// TIA Portal project "ISA_P8" (V16)

(* hardware
DEVICE "S7-1200 station_1"  S7-1200 Station
   slot 0: "Rack_0"  S7-1200 Rack  Rack  V1.0
   slot 1: "PLC_1"  CPU 1215C DC/DC/DC  6ES7 215-1AG40-0XB0  V4.4
DEVICE "PC-System_1"  SIMATIC PC station
   slot 0: "Estación PC SIMATIC"  Rail  SIMATIC PC-Station  V1.0
      slot 125: "Stationmanager"  Station_Manager  V6.0.4
   slot 1: "HMI_RT_1"  WinCC RT Advanced  6AV2 104-0xxxx-xxxx  16.0.0.0
      slot 33792: "Interfaz del equipo"  Host interface
   slot 2: "IE general_1"  IE General  IE_CP  V8.2.0
*)

// ===== PLC "PLC_1"  CPU 1215C DC/DC/DC =====

VAR_GLOBAL   // PLC tag table "Tabla de variables estándar"
   "Pt100" AT %IW64 : Int;   // Entrada Pt100 en bits
   "System_Byte" AT %MB1 : Byte;
   "FirstScan" AT %M1.0 : Bool;
   "DiagStatusUpdate" AT %M1.1 : Bool;
   "AlwaysTRUE" AT %M1.2 : Bool;
   "AlwaysFALSE" AT %M1.3 : Bool;
   "System_Byte(1)" AT %MB1 : Byte;
   "Pulsador Marcha" AT %I0.0 : Bool;
   "Pulsador Paro" AT %I0.1 : Bool;
   "Resistencia" AT %QW64 : Int;
   "Ventilador" AT %Q0.0 : Bool;
   "Selector_Salida_PID" AT %Q0.1 : Bool;
   "Salida_PWM_PID" AT %Q0.2 : Bool;
END_VAR

DATA_BLOCK "IN_Pt100"   // DB1
{ S7_Optimized_Access := 'TRUE' }
VERSION : 0.1
// stored: InstanceOfName Analog_IN
"Analog_IN"
BEGIN
END_DATA_BLOCK

DATA_BLOCK "Variables"   // DB2
{ S7_Optimized_Access := 'TRUE' }
VERSION : 0.1
   VAR
      Temperatura_Pt100 : Real;   // Temperatura Pt100 en ºC
      Modo_PID : Int;   // Modo de funcionamiento del PID
      Mode_Activate : Bool;   // Activación del modo de funcionamiento del PID
      Flanco_Activate : Bool;   // Flanco de "Mode_Activate"
      Flanco_Paro : Bool;   // Flanco de "Pulsador_Paro"
      Reset_PID : Bool;   // Reset del PID en SCADA
      Salida_PID : Real;   // Salida del PID (0-100)
      Setpoint_PID : Real;   // Setpoint del PID
      Ventilador_SCADA : Bool;   // Activación del ventilador desde SCADA
      Mode_Activate_SCADA : Bool;   // Mode_Activate desde SCADA
      State_PID : Int;   // Modo Activo en el PID
      Error_PID : Bool;   // Indicación de error en PID
      Manual_Value_PID : Real;   // Valor manual PID
      ErrorBits_PID : DWord;   // Código de error PID
      Activar_PWM_SCADA : Bool;
      Salida_PWM_SCADA : Real;
      Salida_PWM_PID : Bool;
      Control_Todo_Nada_On : Bool;
      Salida_Control_TN : Bool;
   END_VAR
BEGIN
END_DATA_BLOCK

DATA_BLOCK "Analog_OUT_DB"   // DB4
{ S7_Optimized_Access := 'TRUE' }
VERSION : 0.1
// stored: InstanceOfName Analog_OUT
"Analog_OUT"
BEGIN
END_DATA_BLOCK

DATA_BLOCK "OUT_Resistencia"   // DB5
{ S7_Optimized_Access := 'TRUE' }
VERSION : 0.1
// stored: InstanceOfName Analog_OUT
"Analog_OUT"
BEGIN
END_DATA_BLOCK

DATA_BLOCK "Telerruptor_DB"   // DB6
{ S7_Optimized_Access := 'TRUE' }
VERSION : 0.1
// stored: InstanceOfName Telerruptor
"Telerruptor"
BEGIN
END_DATA_BLOCK

FUNCTION_BLOCK "Telerruptor"   // FB2, LAD
{ S7_Optimized_Access := 'TRUE' }
VERSION : 0.1
   VAR_INPUT
      Pulsador : Bool;
   END_VAR
   VAR_OUTPUT
      Salida : Bool;
   END_VAR
   VAR
      Flanco : Bool;
      "on/off" : Bool;
      state : Bool;
   END_VAR
   VAR_TEMP   // added for the SCL form of the ladder/FBD networks
      _w1 : Bool;
   END_VAR
BEGIN

REGION Network 1
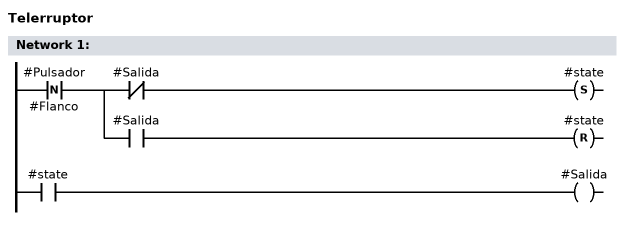
   RUNG wire#powerrail
      N_Contact(operand := #Pulsador, bit := #Flanco)
      wire#w1
      I_Contact( #Salida )
      S_Coil( #state )
   END_RUNG
   RUNG wire#w1
      Contact( #Salida )
      R_Coil( #state )
   END_RUNG
   RUNG wire#powerrail
      Contact( #state )
      Coil( #Salida )
   END_RUNG
   // the same network as SCL:
   #_w1 := NOT #Pulsador AND #Flanco;   // falling edge of #Pulsador
   #Flanco := #Pulsador;
   IF #_w1 AND NOT #Salida THEN #state := TRUE; END_IF;
   IF #_w1 AND #Salida THEN #state := FALSE; END_IF;
   #Salida := #state;
END_REGION
END_FUNCTION_BLOCK

FUNCTION_BLOCK "Analog_IN"   // FB4, LAD
{ S7_Optimized_Access := 'TRUE' }
VERSION : 0.1
   VAR_INPUT
      Input : Int;
      X_min : Real;
      X_max : Real;
      Y_min : Real;
      Y_max : Real;
      IsTension : Bool;
   END_VAR
   VAR_OUTPUT
      Output : Real;
   END_VAR
   VAR
      X_min_bits : Int;
      X_max_bits : Int;
      norm : Real;
   END_VAR
   VAR CONSTANT
      tension_pendent : Real := 2764.8;
      intensity_pendent : Real := 1382.4;
   END_VAR
BEGIN

REGION Network 1 (SCL)

   IF #IsTension THEN
       #X_min_bits := REAL_TO_INT(#X_min * #tension_pendent);
       #X_max_bits := REAL_TO_INT(#X_max * #tension_pendent);
   ELSE
       #X_min_bits := REAL_TO_INT(#X_min * #intensity_pendent);
       #X_max_bits := REAL_TO_INT(#X_max * #intensity_pendent);
   END_IF;
END_REGION

REGION Network 2
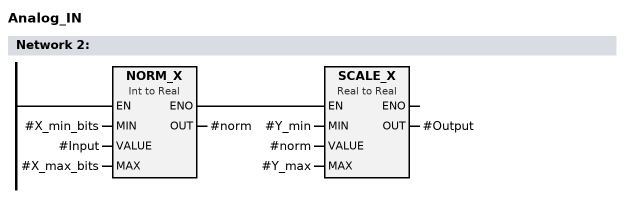
   RUNG wire#powerrail
      { S7_Templates := "[SrcType := Int, DestType := Real]" } Normalize(min := #X_min_bits, value := #Input, max := #X_max_bits, out => #norm)
      { S7_Templates := "[SrcType := Real, DestType := Real]" } Scale(min := #Y_min, value := #norm, max := #Y_max, out => #Output)
   END_RUNG
   // the same network as SCL:
   #norm := NORM_X(MIN := #X_min_bits, VALUE := #Input, MAX := #X_max_bits);
   #Output := SCALE_X(MIN := #Y_min, VALUE := #norm, MAX := #Y_max);
END_REGION
END_FUNCTION_BLOCK

FUNCTION_BLOCK "Analog_OUT"   // FB5, LAD
{ S7_Optimized_Access := 'TRUE' }
VERSION : 0.1
   VAR_INPUT
      Input : Real;
      X_min : Real;
      X_max : Real;
      Y_min : Real;
      Y_max : Real;
      IsTension : Bool;
   END_VAR
   VAR_OUTPUT
      Output : Int;
   END_VAR
   VAR
      Y_min_bits : Int;
      Y_max_bits : Int;
      norm : Real;
   END_VAR
   VAR CONSTANT
      tension_pendent : Real := 2764.8;
      intensity_pendent : Real := 1382.4;
   END_VAR
BEGIN

REGION Network 1 (SCL)

   IF #IsTension THEN
       #Y_min_bits := REAL_TO_INT(#Y_min * #tension_pendent);
       #Y_max_bits := REAL_TO_INT(#Y_max * #tension_pendent);
   ELSE
       #Y_min_bits := REAL_TO_INT(#Y_min * #intensity_pendent);
       #Y_max_bits := REAL_TO_INT(#Y_max * #intensity_pendent);
   END_IF;
END_REGION

REGION Network 2
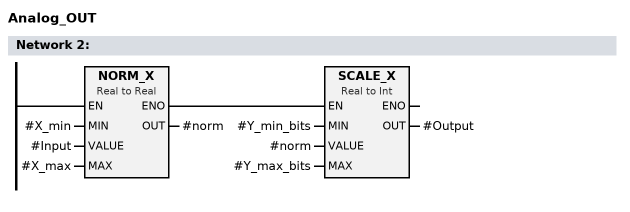
   RUNG wire#powerrail
      { S7_Templates := "[SrcType := Real, DestType := Real]" } Normalize(min := #X_min, value := #Input, max := #X_max, out => #norm)
      { S7_Templates := "[SrcType := Real, DestType := Int]" } Scale(min := #Y_min_bits, value := #norm, max := #Y_max_bits, out => #Output)
   END_RUNG
   // the same network as SCL:
   #norm := NORM_X(MIN := #X_min, VALUE := #Input, MAX := #X_max);
   #Output := SCALE_X(MIN := #Y_min_bits, VALUE := #norm, MAX := #Y_max_bits);
END_REGION
END_FUNCTION_BLOCK

ORGANIZATION_BLOCK "Escalados"   // OB1, LAD, ProgramCycle
TITLE = "Main Program Sweep (Cycle)"
{ S7_Optimized_Access := 'TRUE' }
VERSION : 0.1
   VAR_INPUT
      Initial_Call : Bool;   // Initial call of this OB
      Remanence : Bool;   // =True, if remanent data are available
   END_VAR
BEGIN

REGION Network 1: Escalado acondicionador Pt100
   // Entrada 0-10V del acondicionador de la Pt100 para un rango de 0-100ºC
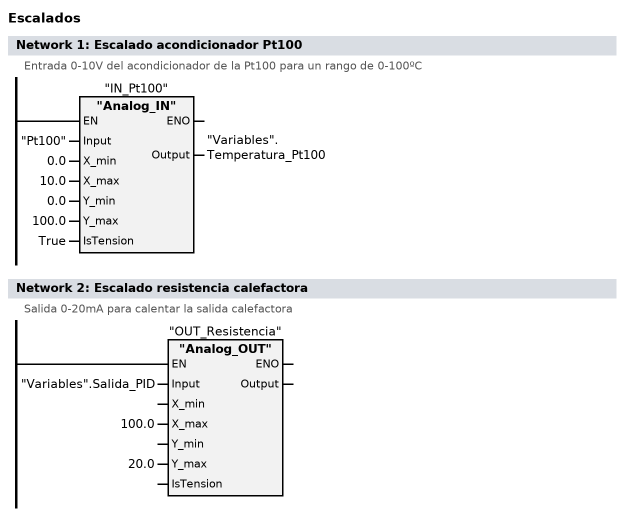
   RUNG wire#powerrail
      "IN_Pt100"(Input := "Pt100", X_min := 0.0, X_max := 10.0, Y_min := 0.0, Y_max := 100.0, IsTension := True, Output => "Variables".Temperatura_Pt100)
   END_RUNG
   // the same network as SCL:
   "IN_Pt100"(Input := "Pt100",   // "Analog_IN"
              X_min := 0.0,
              X_max := 10.0,
              Y_min := 0.0,
              Y_max := 100.0,
              IsTension := True,
              Output => "Variables".Temperatura_Pt100);
END_REGION

REGION Network 2: Escalado resistencia calefactora
   // Salida 0-20mA para calentar la salida calefactora
   RUNG wire#powerrail
      "OUT_Resistencia"(Input := "Variables".Salida_PID, X_min :=, X_max := 100.0, Y_min :=, Y_max := 20.0, IsTension :=, Output =>)
   END_RUNG
   // the same network as SCL:
   "OUT_Resistencia"(Input := "Variables".Salida_PID, X_max := 100.0, Y_max := 20.0);   // "Analog_OUT"
END_REGION

REGION Network 3 (SCL)
   IF "Variables".Salida_PWM_PID THEN
       "Variables".Salida_PWM_SCADA := 100.0;
   ELSE
       "Variables".Salida_PWM_SCADA := 0.0;
   END_IF;
END_REGION
END_ORGANIZATION_BLOCK

ORGANIZATION_BLOCK "PID"   // OB30, LAD, CyclicInterrupt
{ S7_Optimized_Access := 'TRUE' }
VERSION : 0.1
   VAR_INPUT
      Initial_Call : Bool;   // Initial call of this OB
      Event_Count : Int;   // Events discarded
   END_VAR
   VAR_TEMP   // added for the SCL form of the ladder/FBD networks
      _w1 : Bool;
   END_VAR
BEGIN

REGION Network 1: PID
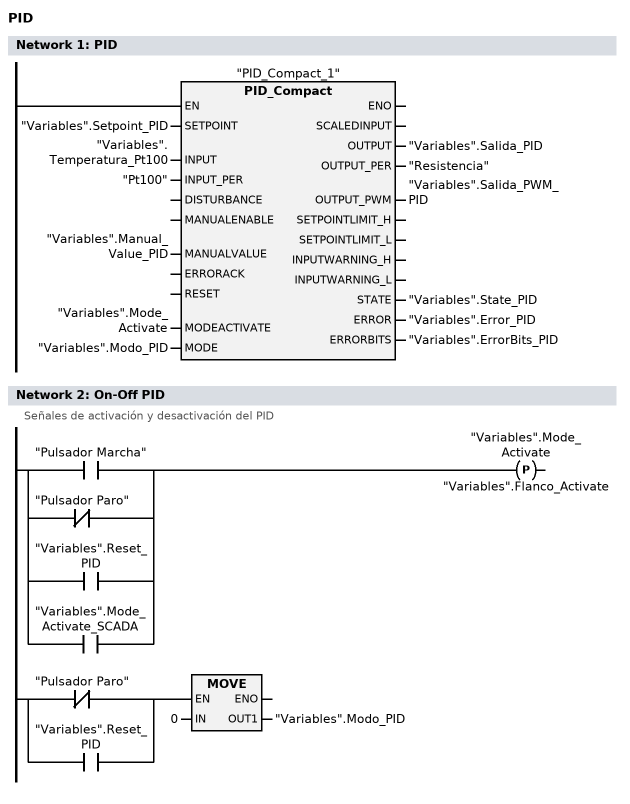
   "PID_Compact_1"(Setpoint := "Variables".Setpoint_PID,   // PID_Compact
                   Input := "Variables".Temperatura_Pt100,
                   Input_PER := "Pt100",
                   ManualValue := "Variables".Manual_Value_PID,
                   ModeActivate := "Variables".Mode_Activate,
                   Mode := "Variables".Modo_PID,
                   Output => "Variables".Salida_PID,
                   Output_PER => "Resistencia",
                   Output_PWM => "Variables".Salida_PWM_PID,
                   State => "Variables".State_PID,
                   Error => "Variables".Error_PID,
                   ErrorBits => "Variables".ErrorBits_PID);
END_REGION

REGION Network 2: On-Off PID
   // Señales de activación y desactivación del PID
   #_w1 := "Pulsador Marcha" OR NOT "Pulsador Paro" OR "Variables".Reset_PID OR "Variables".Mode_Activate_SCADA;
   "Variables".Mode_Activate := #_w1 AND NOT "Variables".Flanco_Activate;   // rising edge
   "Variables".Flanco_Activate := #_w1;
   IF NOT "Pulsador Paro" OR "Variables".Reset_PID THEN "Variables".Modo_PID := 0; END_IF;
END_REGION

REGION Network 3 (SCL)
   "PID_Compact_1".Config.InputPerOn := TRUE;
END_REGION
END_ORGANIZATION_BLOCK

ORGANIZATION_BLOCK "Salidas"   // OB123, LAD, ProgramCycle
TITLE = "Main Program Sweep (Cycle)"
{ S7_Optimized_Access := 'TRUE' }
VERSION : 0.1
   VAR_INPUT
      Initial_Call : Bool;   // Initial call of this OB
      Remanence : Bool;   // =True, if remanent data are available
   END_VAR
BEGIN

REGION Network 1: On-Off Ventilador
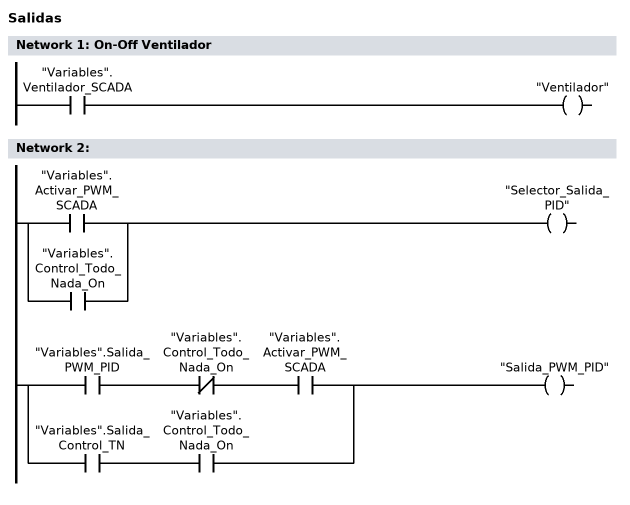
   RUNG wire#powerrail
      Contact( "Variables".Ventilador_SCADA )
      Coil( "Ventilador" )
   END_RUNG
   // the same network as SCL:
   "Ventilador" := "Variables".Ventilador_SCADA;
END_REGION

REGION Network 2
   RUNG wire#powerrail
      Contact( "Variables".Activar_PWM_SCADA )
      wire#w1
      Coil( "Selector_Salida_PID" )
   END_RUNG
   RUNG wire#powerrail
      Contact( "Variables".Control_Todo_Nada_On )
   END_RUNG wire#w1
   RUNG wire#powerrail
      Contact( "Variables".Salida_PWM_PID )
      I_Contact( "Variables".Control_Todo_Nada_On )
      Contact( "Variables".Activar_PWM_SCADA )
      wire#w2
      Coil( "Salida_PWM_PID" )
   END_RUNG
   RUNG wire#powerrail
      Contact( "Variables".Salida_Control_TN )
      Contact( "Variables".Control_Todo_Nada_On )
   END_RUNG wire#w2
   // the same network as SCL:
   "Selector_Salida_PID" := "Variables".Activar_PWM_SCADA OR "Variables".Control_Todo_Nada_On;
   "Salida_PWM_PID" := ("Variables".Salida_PWM_PID AND NOT "Variables".Control_Todo_Nada_On AND "Variables".Activar_PWM_SCADA) OR ("Variables".Salida_Control_TN AND "Variables".Control_Todo_Nada_On);
END_REGION
END_ORGANIZATION_BLOCK

ORGANIZATION_BLOCK "Control_Todo_Nada"   // OB124, SCL, ProgramCycle
TITLE = "Main Program Sweep (Cycle)"
{ S7_Optimized_Access := 'TRUE' }
VERSION : 0.1
   VAR_INPUT
      Initial_Call : Bool;   // Initial call of this OB
      Remanence : Bool;   // =True, if remanent data are available
   END_VAR
BEGIN
   IF "Variables".Temperatura_Pt100 >= "Variables".Setpoint_PID THEN
       "Variables".Salida_Control_TN := FALSE;
   ELSE
       "Variables".Salida_Control_TN := TRUE;
   END_IF;
END_ORGANIZATION_BLOCK

(* ===== HMI "HMI_RT_1" =====
system functions are stored by id; their names below are inferred from use
connection "HMI_Conexión_1": ETHERNET, S7_1200_OMS

HMI tags "Tabla de variables estándar"
   "Variables_Temperatura_Pt100" : Real = PLC Variables.Temperatura_Pt100, 1 s
   "Variables_Modo_PID" : Int = PLC Variables.Modo_PID, 1 s
   "Variables_Ventilador_SCADA" : Bool = PLC Variables.Ventilador_SCADA, 1 s
   "Variables_Setpoint_PID" : Real = PLC Variables.Setpoint_PID, 1 s
   "Variables_Mode_Activate_SCADA" : Bool = PLC Variables.Mode_Activate_SCADA, 1 s
   "Variables_Reset_PID" : Bool = PLC Variables.Reset_PID, 1 s
   "Variables_Salida_PID" : Real = PLC Variables.Salida_PID, 1 s
   "Variables_Error_PID" : Bool = PLC Variables.Error_PID, 1 s
   "Variables_Manual_Value_PID" : Real = PLC Variables.Manual_Value_PID, 1 s
   "Variables_State_PID" : Int = PLC Variables.State_PID, 1 s
   "Variables_ErrorBits_PID" : DWord = PLC Variables.ErrorBits_PID, 1 s
   "PID_Compact_1_Retain_CtrlParams_Gain" : Real = PLC PID_Compact_1.Retain.CtrlParams.Gain, 1 s
   "PID_Compact_1_Retain_CtrlParams_Ti" : Real = PLC PID_Compact_1.Retain.CtrlParams.Ti, 1 s
   "PID_Compact_1_Retain_CtrlParams_Td" : Real = PLC PID_Compact_1.Retain.CtrlParams.Td, 1 s
   "Variables_Activar_PWM_SCADA" : Bool = PLC Variables.Activar_PWM_SCADA, 1 s
   "Variables_Salida_PWM_SCADA" : Real = PLC Variables.Salida_PWM_SCADA, 1 s
   "PID_Compact_1_Retain_CtrlParams_Cycle" : Real = PLC PID_Compact_1.Retain.CtrlParams.Cycle, 1 s
   "PID_Compact_1_Config_MinimumOnTime" : Real = PLC PID_Compact_1.Config.MinimumOnTime, 1 s
   "PID_Compact_1_Config_MinimumOffTime" : Real = PLC PID_Compact_1.Config.MinimumOffTime, 1 s
   "Variables_Control_Todo_Nada_On" : Bool = PLC Variables.Control_Todo_Nada_On, 1 s

text list "Modos_PID": 1 'Optimización Inicial'; 2 'Optimización Fina Manual'; 3 'Modo Automático'; 4 'Modo Manual'

screen "Imagen_1" 800x600
   IOField "Campo ES_1" at 140,209 size 96x32; FormatPattern 999.99; Unit ºC
      ProcessValue <- "Variables_Temperatura_Pt100"
   SymbolicIOField "Campo ES simbólico_1" at 26,530 size 216x32; TextOff '0'; TextOn '1'; TextList "Modos_PID"
      ProcessValue <- "Variables_Modo_PID"
   GraphicView "Visor de gráficos_1" at 254,33 size 251x520; Picture "Captura de pantalla 2023-12-13 131257"
   IOField "Campo ES_2" at 140,123 size 96x32; FormatPattern 99.99
      ProcessValue <- "Variables_Setpoint_PID"
   Button "Botón_1" at 111,42 size 121x32; TextOff 'Ventilador'
      on Click: InvertBit("Variables_Ventilador_SCADA")
   Button "Botón_3" at 146,471 size 96x32; TextOff 'Activate'
      on Press: SetBit("Variables_Mode_Activate_SCADA")
      on Release: ResetBit("Variables_Mode_Activate_SCADA")
   Button "Botón_2" at 26,471 size 96x32; TextOff 'Stop'
      on Press: SetBit("Variables_Reset_PID")
      on Release: ResetBit("Variables_Reset_PID")
   IOField "Campo ES_3" at 519,177 size 96x32; FormatPattern 999.99
      ProcessValue <- "Variables_Salida_PID"
   IOField "Campo ES_4" at 519,400 size 96x32; FormatPattern 9
      ProcessValue <- "Variables_State_PID"
   Rectangle "Rectángulo_1" at 518,436 size 96x20
      Appearance <- "Variables_Error_PID"
   IOField "Campo ES_5" at 140,325 size 96x32; FormatPattern 999.99
      ProcessValue <- "Variables_Manual_Value_PID"
   IOField "Campo ES_6" at 653,25 size 96x32; FormatPattern 99.99
      ProcessValue <- "PID_Compact_1_Retain_CtrlParams_Gain"
   TextField "Campo de texto_1" at 620,29 size 22x22; Text 'k'
   Button "Botón_4" at 652,541 size 96x32; TextOff 'Gráficos'
      on Click: ActivateScreen("Imagen_2", 0)
   IOField "Campo ES_7" at 653,74 size 96x32; FormatPattern 999.99
      ProcessValue <- "PID_Compact_1_Retain_CtrlParams_Ti"
   TextField "Campo de texto_2" at 620,78 size 30x22; Text 'Ti'
   IOField "Campo ES_8" at 653,123 size 96x32; FormatPattern 99.99
      ProcessValue <- "PID_Compact_1_Retain_CtrlParams_Td"
   TextField "Campo de texto_3" at 620,127 size 31x22; Text 'Td'
   IOField "Campo ES_9" at 518,462 size 98x32; FormatPattern FFFF
      ProcessValue <- "Variables_ErrorBits_PID"
   Switch "Interruptor_1" at 642,214 size 120x88; CaptionText 'Salida PWM'; TextOff 'OFF'; TextOn 'ON'
      ProcessValue <- "Variables_Activar_PWM_SCADA"
   IOField "Campo ES_10" at 651,353 size 96x32; FormatPattern 99.99
      ProcessValue <- "PID_Compact_1_Retain_CtrlParams_Cycle"
   TextField "Campo de texto_4" at 605,325 size 169x22; Text 'Tiempo Algoritmo'
   IOField "Campo ES_11" at 651,420 size 96x32; FormatPattern 99.99
      ProcessValue <- "PID_Compact_1_Config_MinimumOnTime"
   TextField "Campo de texto_5" at 656,393 size 132x22; Text 'T_On'
   IOField "Campo ES_12" at 651,487 size 96x32; FormatPattern 99.99
      ProcessValue <- "PID_Compact_1_Config_MinimumOffTime"
   TextField "Campo de texto_6" at 656,460 size 132x22; Text 'T_Off'
   Button "Botón_5" at 17,178 size 96x32; TextOff 'inicio file'
      on Click: function_fd9437ed(0, "PID")
   Button "Botón_6" at 17,223 size 96x32; TextOff 'paro file'
      on Click: function_b6526003(0, "PID")
   Switch "Interruptor_2" at 26,357 size 120x88; TextOn 'ON'; CaptionText 'TODO/NADA'; TextOff 'OFF'
      ProcessValue <- "Variables_Control_Todo_Nada_On"

screen "Imagen_2" 800x600
   Button "Botón_4" at 652,541 size 96x32; TextOff 'Control'
      on Click: ActivateScreen("Imagen_1", 0)
   TrendView "Visor de curvas_1" at 90,45 size 600x462
*)